Universal Robots PolyScope program: ryan_test_2.urp

Program ryan_test_2 (installation=default directory=/programs createdIn=5.9.1.1031110 lastSavedIn=5.9.1.1031110 robotSerialNumber=20195501059)
Calibrated DH parameters: a=[0.000146, -0.418764, -0.053981, 0.000058, -0.000023, 0]; d=[0.162545, 37.319448, -206.067439, 168.881546, 0.09955, 0.099464]; alpha=[1.57004, -0.001979, 0.002304, 1.570607, -1.57066, 0]; deltaTheta=[0, -0.174616, -1.258233, 1.432844, -0.000001, 0]
Robot Program (runOnlyOnce=false)
  MoveL speed 250 mm/s, acceleration 1200 mm/s^2 (useActiveTCP=true) feature=Base
    Waypoint Waypoint_1: TCP in base x=374.572 y=-191.849 z=57.853 mm, rx=-2.2213 ry=-2.1997 rz=0.0166 rad; joints [134.781, -89.167, 129.618, -129.562, 269.465, 135.378] deg; TCP offset x=0 y=0 z=174 mm, rx=0 ry=0 rz=0 rad
    Waypoint Waypoint_2: TCP in base x=374.577 y=-191.843 z=154.076 mm, rx=-2.2213 ry=-2.1997 rz=0.0166 rad; joints [134.786, -97.549, 120.783, -112.342, 269.453, 135.355] deg
    Waypoint Waypoint_1: TCP in base x=374.572 y=-191.849 z=57.853 mm, rx=-2.2213 ry=-2.1997 rz=0.0166 rad; joints [134.781, -89.167, 129.618, -129.562, 269.465, 135.378] deg
